DATA_BLOCK "Simulace"
{ S7_Optimized_Access := 'TRUE' }
VERSION : 0.1
NON_RETAIN
   VAR
      Timer_Simulace {InstructionName := 'IEC_TIMER'; LibVersion := '1.0'; S7_SetPoint := 'False'} : IEC_TIMER;
      Source_Cell { S7_SetPoint := 'True'} : Int;
      Target_Cell : Int;
      Set_time_simulace { S7_SetPoint := 'True'} : Time;   // nastaveni doby trvani simulace
      TransportMatrix : Array[1..6, 1..6] of Int;
      Sim_start { S7_SetPoint := 'True'} : Bool;
      Sim_end : Bool;
      run_time : Time;
      Sim_BTN : Bool;
      State_Int : Int;
   END_VAR


BEGIN
   TransportMatrix[1,2] := 8;
   TransportMatrix[1,3] := 6;
   TransportMatrix[1,4] := 3;
   TransportMatrix[1,5] := 7;
   TransportMatrix[1,6] := 2;
   TransportMatrix[2,1] := 8;
   TransportMatrix[2,2] := 0;
   TransportMatrix[2,3] := 3;
   TransportMatrix[2,4] := 6;
   TransportMatrix[2,5] := 2;
   TransportMatrix[2,6] := 7;
   TransportMatrix[3,1] := 6;
   TransportMatrix[3,2] := 3;
   TransportMatrix[3,3] := 0;
   TransportMatrix[3,4] := 4;
   TransportMatrix[3,5] := 2;
   TransportMatrix[3,6] := 5;
   TransportMatrix[4,1] := 3;
   TransportMatrix[4,2] := 6;
   TransportMatrix[4,3] := 4;
   TransportMatrix[4,4] := 0;
   TransportMatrix[4,5] := 5;
   TransportMatrix[4,6] := 2;
   TransportMatrix[5,1] := 7;
   TransportMatrix[5,2] := 2;
   TransportMatrix[5,3] := 2;
   TransportMatrix[5,4] := 5;
   TransportMatrix[5,5] := 0;
   TransportMatrix[5,6] := 8;
   TransportMatrix[6,1] := 2;
   TransportMatrix[6,2] := 7;
   TransportMatrix[6,3] := 5;
   TransportMatrix[6,4] := 2;
   TransportMatrix[6,5] := 8;

END_DATA_BLOCK

